// TIA Portal V20 export
FUNCTION "CollectAlarms" : Void   // FC91, LAD
TITLE = Alarm Collector Unit
// Collects alarms from the respective level and categorises the alarms into the different alarm classes.
// stored: Namespace Unit1.Em5, SetENOAutomatically false
   VAR_INPUT
      resetAlarms : Bool;
      disableAlarms : Bool;
   END_VAR
   VAR_OUTPUT
      commandsToUnit : "LUC_typeStateCommands";   // Feedback to the unit
   END_VAR
   VAR CONSTANT
      DelayTime : Time := T#300ms;
      TRUE : Bool := TRUE;
      FALSE : Bool := FALSE;
   END_VAR
BEGIN

REGION Network 1: Reset Alarms
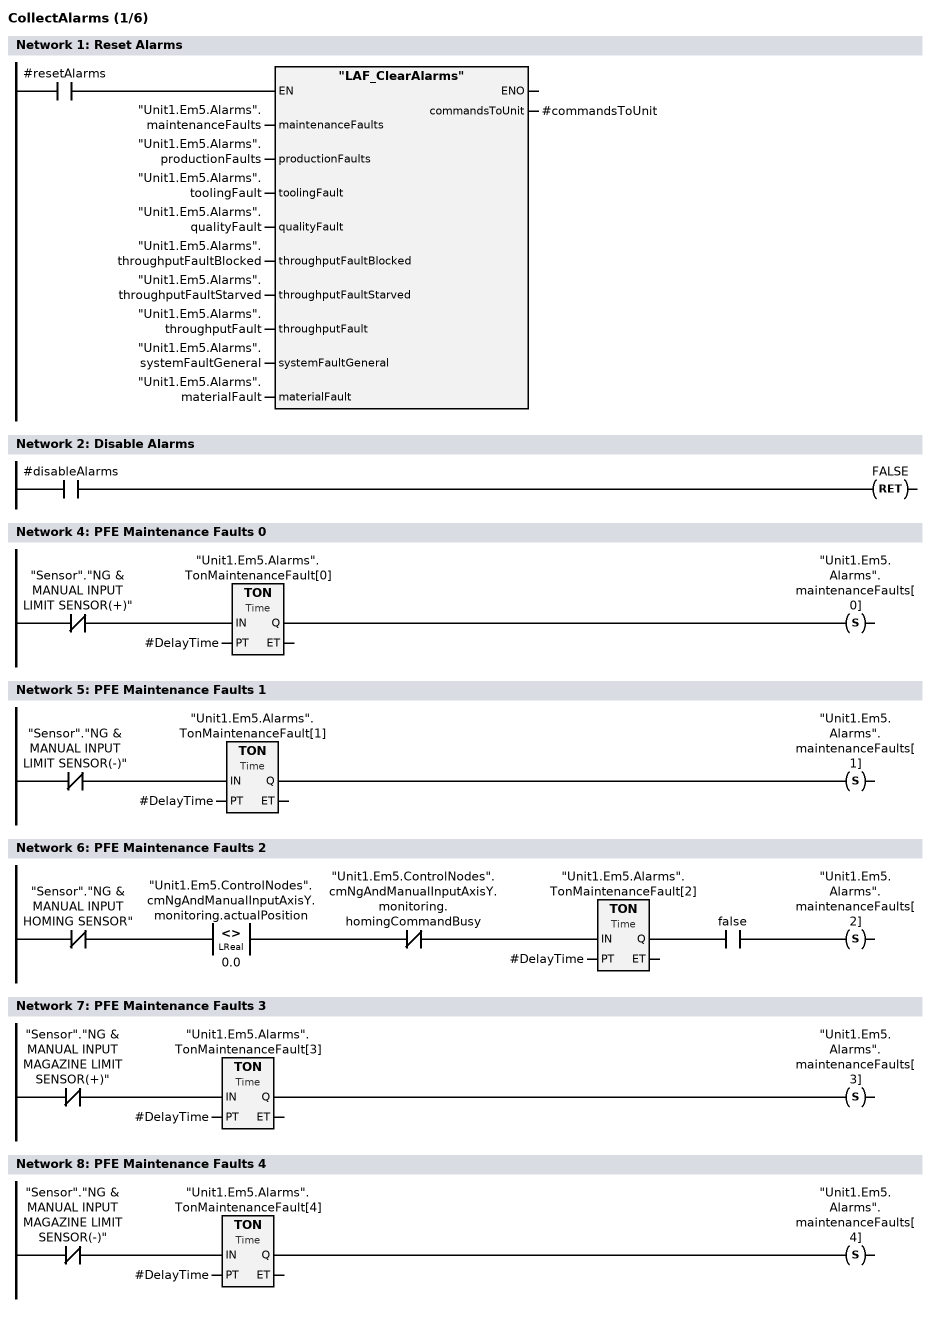
   RUNG wire#powerrail
      Contact( #resetAlarms )
      "LAF_ClearAlarms"(maintenanceFaults := "Unit1.Em5.Alarms".maintenanceFaults, productionFaults := "Unit1.Em5.Alarms".productionFaults, toolingFault := "Unit1.Em5.Alarms".toolingFault, qualityFault := "Unit1.Em5.Alarms".qualityFault, throughputFaultBlocked := "Unit1.Em5.Alarms".throughputFaultBlocked, throughputFaultStarved := "Unit1.Em5.Alarms".throughputFaultStarved, throughputFault := "Unit1.Em5.Alarms".throughputFault, systemFaultGeneral := "Unit1.Em5.Alarms".systemFaultGeneral, materialFault := "Unit1.Em5.Alarms".materialFault, commandsToUnit => #commandsToUnit)
   END_RUNG
   // the same network as SCL:
   IF #resetAlarms THEN
       "LAF_ClearAlarms"(maintenanceFaults := "Unit1.Em5.Alarms".maintenanceFaults,
                         productionFaults := "Unit1.Em5.Alarms".productionFaults,
                         toolingFault := "Unit1.Em5.Alarms".toolingFault,
                         qualityFault := "Unit1.Em5.Alarms".qualityFault,
                         throughputFaultBlocked := "Unit1.Em5.Alarms".throughputFaultBlocked,
                         throughputFaultStarved := "Unit1.Em5.Alarms".throughputFaultStarved,
                         throughputFault := "Unit1.Em5.Alarms".throughputFault,
                         systemFaultGeneral := "Unit1.Em5.Alarms".systemFaultGeneral,
                         materialFault := "Unit1.Em5.Alarms".materialFault,
                         commandsToUnit => #commandsToUnit);
   END_IF;
END_REGION

REGION Network 2: Disable Alarms
   RUNG wire#powerrail
      Contact( #disableAlarms )
      ReturnCoil( FALSE )
   END_RUNG
   // the same network as SCL:
   IF #disableAlarms THEN
       ENO := FALSE;
       RETURN;
   END_IF;
END_REGION

REGION Network 3: *************** Fault ************************
END_REGION

REGION Network 4: PFE Maintenance Faults 0
   RUNG wire#powerrail
      I_Contact( "Sensor"."NG & MANUAL INPUT LIMIT SENSOR(+)" )
      { S7_Templates := "time_type := Time" } "Unit1.Em5.Alarms".TonMaintenanceFault[0].TON(pt := #DelayTime, et =>)
      S_Coil( "Unit1.Em5.Alarms".maintenanceFaults[0] )
   END_RUNG
   // the same network as SCL:
   "Unit1.Em5.Alarms".TonMaintenanceFault[0].TON(IN := NOT "Sensor"."NG & MANUAL INPUT LIMIT SENSOR(+)",
                           PT := #DelayTime);
   IF "Unit1.Em5.Alarms".TonMaintenanceFault[0].Q THEN
       "Unit1.Em5.Alarms".maintenanceFaults[0] := TRUE;
   END_IF;
END_REGION

REGION Network 5: PFE Maintenance Faults 1
   RUNG wire#powerrail
      I_Contact( "Sensor"."NG & MANUAL INPUT LIMIT SENSOR(-)" )
      { S7_Templates := "time_type := Time" } "Unit1.Em5.Alarms".TonMaintenanceFault[1].TON(pt := #DelayTime, et =>)
      S_Coil( "Unit1.Em5.Alarms".maintenanceFaults[1] )
   END_RUNG
   // the same network as SCL:
   "Unit1.Em5.Alarms".TonMaintenanceFault[1].TON(IN := NOT "Sensor"."NG & MANUAL INPUT LIMIT SENSOR(-)",
                           PT := #DelayTime);
   IF "Unit1.Em5.Alarms".TonMaintenanceFault[1].Q THEN
       "Unit1.Em5.Alarms".maintenanceFaults[1] := TRUE;
   END_IF;
END_REGION

REGION Network 6: PFE Maintenance Faults 2
   RUNG wire#powerrail
      I_Contact( "Sensor"."NG & MANUAL INPUT HOMING SENSOR" )
      { S7_Templates := "SrcType := LReal" } NE_Contact(in1 := "Unit1.Em5.ControlNodes".cmNgAndManualInputAxisY.monitoring.actualPosition, in2 := 0.0)
      I_Contact( "Unit1.Em5.ControlNodes".cmNgAndManualInputAxisY.monitoring.homingCommandBusy )
      { S7_Templates := "time_type := Time" } "Unit1.Em5.Alarms".TonMaintenanceFault[2].TON(pt := #DelayTime, et =>)
      Contact( false )
      S_Coil( "Unit1.Em5.Alarms".maintenanceFaults[2] )
   END_RUNG
   // the same network as SCL:
   "Unit1.Em5.Alarms".TonMaintenanceFault[2].TON(IN := NOT "Sensor"."NG & MANUAL INPUT HOMING SENSOR" AND ("Unit1.Em5.ControlNodes".cmNgAndManualInputAxisY.monitoring.actualPosition <> 0.0) AND NOT "Unit1.Em5.ControlNodes".cmNgAndManualInputAxisY.monitoring.homingCommandBusy,
                           PT := #DelayTime);
   IF "Unit1.Em5.Alarms".TonMaintenanceFault[2].Q AND false THEN
       "Unit1.Em5.Alarms".maintenanceFaults[2] := TRUE;
   END_IF;
END_REGION

REGION Network 7: PFE Maintenance Faults 3
   RUNG wire#powerrail
      I_Contact( "Sensor"."NG & MANUAL INPUT MAGAZINE LIMIT SENSOR(+)" )
      { S7_Templates := "time_type := Time" } "Unit1.Em5.Alarms".TonMaintenanceFault[3].TON(pt := #DelayTime, et =>)
      S_Coil( "Unit1.Em5.Alarms".maintenanceFaults[3] )
   END_RUNG
   // the same network as SCL:
   "Unit1.Em5.Alarms".TonMaintenanceFault[3].TON(IN := NOT "Sensor"."NG & MANUAL INPUT MAGAZINE LIMIT SENSOR(+)",
                           PT := #DelayTime);
   IF "Unit1.Em5.Alarms".TonMaintenanceFault[3].Q THEN
       "Unit1.Em5.Alarms".maintenanceFaults[3] := TRUE;
   END_IF;
END_REGION

REGION Network 8: PFE Maintenance Faults 4
   RUNG wire#powerrail
      I_Contact( "Sensor"."NG & MANUAL INPUT MAGAZINE LIMIT SENSOR(-)" )
      { S7_Templates := "time_type := Time" } "Unit1.Em5.Alarms".TonMaintenanceFault[4].TON(pt := #DelayTime, et =>)
      S_Coil( "Unit1.Em5.Alarms".maintenanceFaults[4] )
   END_RUNG
   // the same network as SCL:
   "Unit1.Em5.Alarms".TonMaintenanceFault[4].TON(IN := NOT "Sensor"."NG & MANUAL INPUT MAGAZINE LIMIT SENSOR(-)",
                           PT := #DelayTime);
   IF "Unit1.Em5.Alarms".TonMaintenanceFault[4].Q THEN
       "Unit1.Em5.Alarms".maintenanceFaults[4] := TRUE;
   END_IF;
END_REGION

REGION Network 9: PFE Maintenance Faults 5
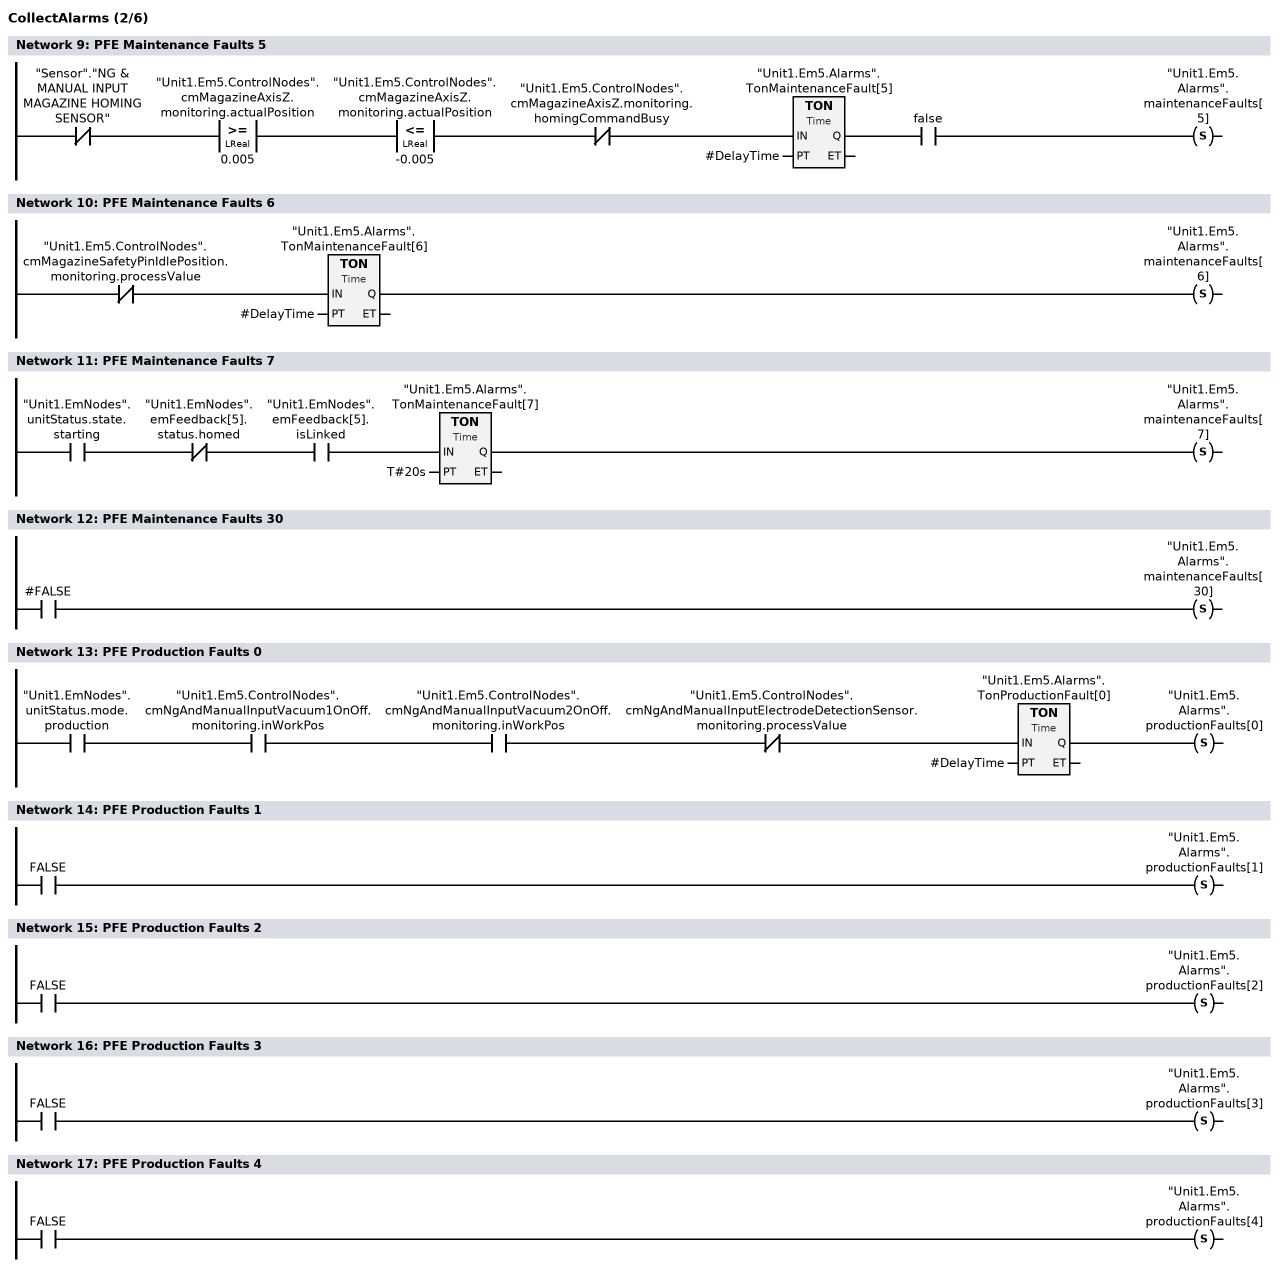
   RUNG wire#powerrail
      I_Contact( "Sensor"."NG & MANUAL INPUT MAGAZINE HOMING SENSOR" )
      { S7_Templates := "SrcType := LReal" } GE_Contact(in1 := "Unit1.Em5.ControlNodes".cmMagazineAxisZ.monitoring.actualPosition, in2 := 0.005)
      { S7_Templates := "SrcType := LReal" } LE_Contact(in1 := "Unit1.Em5.ControlNodes".cmMagazineAxisZ.monitoring.actualPosition, in2 := -0.005)
      I_Contact( "Unit1.Em5.ControlNodes".cmMagazineAxisZ.monitoring.homingCommandBusy )
      { S7_Templates := "time_type := Time" } "Unit1.Em5.Alarms".TonMaintenanceFault[5].TON(pt := #DelayTime, et =>)
      Contact( false )
      S_Coil( "Unit1.Em5.Alarms".maintenanceFaults[5] )
   END_RUNG
   // the same network as SCL:
   "Unit1.Em5.Alarms".TonMaintenanceFault[5].TON(IN := NOT "Sensor"."NG & MANUAL INPUT MAGAZINE HOMING SENSOR" AND ("Unit1.Em5.ControlNodes".cmMagazineAxisZ.monitoring.actualPosition >= 0.005) AND ("Unit1.Em5.ControlNodes".cmMagazineAxisZ.monitoring.actualPosition <= (-0.005)) AND NOT "Unit1.Em5.ControlNodes".cmMagazineAxisZ.monitoring.homingCommandBusy,
                           PT := #DelayTime);
   IF "Unit1.Em5.Alarms".TonMaintenanceFault[5].Q AND false THEN
       "Unit1.Em5.Alarms".maintenanceFaults[5] := TRUE;
   END_IF;
END_REGION

REGION Network 10: PFE Maintenance Faults 6
   RUNG wire#powerrail
      I_Contact( "Unit1.Em5.ControlNodes".cmMagazineSafetyPinIdlePosition.monitoring.processValue )
      { S7_Templates := "time_type := Time" } "Unit1.Em5.Alarms".TonMaintenanceFault[6].TON(pt := #DelayTime, et =>)
      S_Coil( "Unit1.Em5.Alarms".maintenanceFaults[6] )
   END_RUNG
   // the same network as SCL:
   "Unit1.Em5.Alarms".TonMaintenanceFault[6].TON(IN := NOT "Unit1.Em5.ControlNodes".cmMagazineSafetyPinIdlePosition.monitoring.processValue,
                           PT := #DelayTime);
   IF "Unit1.Em5.Alarms".TonMaintenanceFault[6].Q THEN
       "Unit1.Em5.Alarms".maintenanceFaults[6] := TRUE;
   END_IF;
END_REGION

REGION Network 11: PFE Maintenance Faults 7
   RUNG wire#powerrail
      Contact( "Unit1.EmNodes".unitStatus.state.starting )
      I_Contact( "Unit1.EmNodes".emFeedback[5].status.homed )
      Contact( "Unit1.EmNodes".emFeedback[5].isLinked )
      { S7_Templates := "time_type := Time" } "Unit1.Em5.Alarms".TonMaintenanceFault[7].TON(pt := T#20s, et =>)
      S_Coil( "Unit1.Em5.Alarms".maintenanceFaults[7] )
   END_RUNG
   // the same network as SCL:
   "Unit1.Em5.Alarms".TonMaintenanceFault[7].TON(IN := "Unit1.EmNodes".unitStatus.state.starting AND NOT "Unit1.EmNodes".emFeedback[5].status.homed AND "Unit1.EmNodes".emFeedback[5].isLinked,
                           PT := T#20s);
   IF "Unit1.Em5.Alarms".TonMaintenanceFault[7].Q THEN
       "Unit1.Em5.Alarms".maintenanceFaults[7] := TRUE;
   END_IF;
END_REGION

REGION Network 12: PFE Maintenance Faults 30
   RUNG wire#powerrail
      Contact( #FALSE )
      S_Coil( "Unit1.Em5.Alarms".maintenanceFaults[30] )
   END_RUNG
   // the same network as SCL:
   IF #FALSE THEN "Unit1.Em5.Alarms".maintenanceFaults[30] := TRUE; END_IF;
END_REGION

REGION Network 13: PFE Production Faults 0
   RUNG wire#powerrail
      Contact( "Unit1.EmNodes".unitStatus.mode.production )
      Contact( "Unit1.Em5.ControlNodes".cmNgAndManualInputVacuum1OnOff.monitoring.inWorkPos )
      Contact( "Unit1.Em5.ControlNodes".cmNgAndManualInputVacuum2OnOff.monitoring.inWorkPos )
      I_Contact( "Unit1.Em5.ControlNodes".cmNgAndManualInputElectrodeDetectionSensor.monitoring.processValue )
      { S7_Templates := "time_type := Time" } "Unit1.Em5.Alarms".TonProductionFault[0].TON(pt := #DelayTime, et =>)
      S_Coil( "Unit1.Em5.Alarms".productionFaults[0] )
   END_RUNG
   // the same network as SCL:
   "Unit1.Em5.Alarms".TonProductionFault[0].TON(IN := "Unit1.EmNodes".unitStatus.mode.production AND "Unit1.Em5.ControlNodes".cmNgAndManualInputVacuum1OnOff.monitoring.inWorkPos AND "Unit1.Em5.ControlNodes".cmNgAndManualInputVacuum2OnOff.monitoring.inWorkPos AND NOT "Unit1.Em5.ControlNodes".cmNgAndManualInputElectrodeDetectionSensor.monitoring.processValue,
                           PT := #DelayTime);
   IF "Unit1.Em5.Alarms".TonProductionFault[0].Q THEN "Unit1.Em5.Alarms".productionFaults[0] := TRUE; END_IF;
END_REGION

REGION Network 14: PFE Production Faults 1
   RUNG wire#powerrail
      Contact( FALSE )
      S_Coil( "Unit1.Em5.Alarms".productionFaults[1] )
   END_RUNG
   // the same network as SCL:
   IF FALSE THEN "Unit1.Em5.Alarms".productionFaults[1] := TRUE; END_IF;
END_REGION

REGION Network 15: PFE Production Faults 2
   RUNG wire#powerrail
      Contact( FALSE )
      S_Coil( "Unit1.Em5.Alarms".productionFaults[2] )
   END_RUNG
   // the same network as SCL:
   IF FALSE THEN "Unit1.Em5.Alarms".productionFaults[2] := TRUE; END_IF;
END_REGION

REGION Network 16: PFE Production Faults 3
   RUNG wire#powerrail
      Contact( FALSE )
      S_Coil( "Unit1.Em5.Alarms".productionFaults[3] )
   END_RUNG
   // the same network as SCL:
   IF FALSE THEN "Unit1.Em5.Alarms".productionFaults[3] := TRUE; END_IF;
END_REGION

REGION Network 17: PFE Production Faults 4
   RUNG wire#powerrail
      Contact( FALSE )
      S_Coil( "Unit1.Em5.Alarms".productionFaults[4] )
   END_RUNG
   // the same network as SCL:
   IF FALSE THEN "Unit1.Em5.Alarms".productionFaults[4] := TRUE; END_IF;
END_REGION

REGION Network 18: PFE Tooling Faults 0
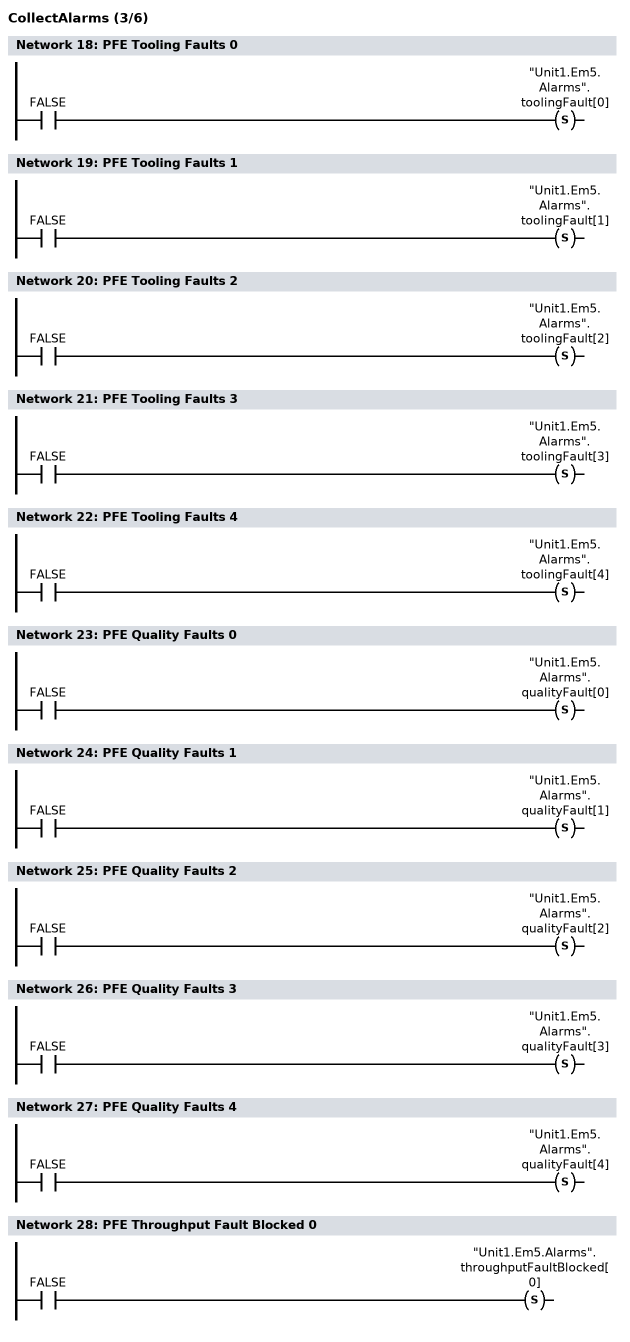
   RUNG wire#powerrail
      Contact( FALSE )
      S_Coil( "Unit1.Em5.Alarms".toolingFault[0] )
   END_RUNG
   // the same network as SCL:
   IF FALSE THEN "Unit1.Em5.Alarms".toolingFault[0] := TRUE; END_IF;
END_REGION

REGION Network 19: PFE Tooling Faults 1
   RUNG wire#powerrail
      Contact( FALSE )
      S_Coil( "Unit1.Em5.Alarms".toolingFault[1] )
   END_RUNG
   // the same network as SCL:
   IF FALSE THEN "Unit1.Em5.Alarms".toolingFault[1] := TRUE; END_IF;
END_REGION

REGION Network 20: PFE Tooling Faults 2
   RUNG wire#powerrail
      Contact( FALSE )
      S_Coil( "Unit1.Em5.Alarms".toolingFault[2] )
   END_RUNG
   // the same network as SCL:
   IF FALSE THEN "Unit1.Em5.Alarms".toolingFault[2] := TRUE; END_IF;
END_REGION

REGION Network 21: PFE Tooling Faults 3
   RUNG wire#powerrail
      Contact( FALSE )
      S_Coil( "Unit1.Em5.Alarms".toolingFault[3] )
   END_RUNG
   // the same network as SCL:
   IF FALSE THEN "Unit1.Em5.Alarms".toolingFault[3] := TRUE; END_IF;
END_REGION

REGION Network 22: PFE Tooling Faults 4
   RUNG wire#powerrail
      Contact( FALSE )
      S_Coil( "Unit1.Em5.Alarms".toolingFault[4] )
   END_RUNG
   // the same network as SCL:
   IF FALSE THEN "Unit1.Em5.Alarms".toolingFault[4] := TRUE; END_IF;
END_REGION

REGION Network 23: PFE Quality Faults 0
   RUNG wire#powerrail
      Contact( FALSE )
      S_Coil( "Unit1.Em5.Alarms".qualityFault[0] )
   END_RUNG
   // the same network as SCL:
   IF FALSE THEN "Unit1.Em5.Alarms".qualityFault[0] := TRUE; END_IF;
END_REGION

REGION Network 24: PFE Quality Faults 1
   RUNG wire#powerrail
      Contact( FALSE )
      S_Coil( "Unit1.Em5.Alarms".qualityFault[1] )
   END_RUNG
   // the same network as SCL:
   IF FALSE THEN "Unit1.Em5.Alarms".qualityFault[1] := TRUE; END_IF;
END_REGION

REGION Network 25: PFE Quality Faults 2
   RUNG wire#powerrail
      Contact( FALSE )
      S_Coil( "Unit1.Em5.Alarms".qualityFault[2] )
   END_RUNG
   // the same network as SCL:
   IF FALSE THEN "Unit1.Em5.Alarms".qualityFault[2] := TRUE; END_IF;
END_REGION

REGION Network 26: PFE Quality Faults 3
   RUNG wire#powerrail
      Contact( FALSE )
      S_Coil( "Unit1.Em5.Alarms".qualityFault[3] )
   END_RUNG
   // the same network as SCL:
   IF FALSE THEN "Unit1.Em5.Alarms".qualityFault[3] := TRUE; END_IF;
END_REGION

REGION Network 27: PFE Quality Faults 4
   RUNG wire#powerrail
      Contact( FALSE )
      S_Coil( "Unit1.Em5.Alarms".qualityFault[4] )
   END_RUNG
   // the same network as SCL:
   IF FALSE THEN "Unit1.Em5.Alarms".qualityFault[4] := TRUE; END_IF;
END_REGION

REGION Network 28: PFE Throughput Fault Blocked 0
   RUNG wire#powerrail
      Contact( FALSE )
      S_Coil( "Unit1.Em5.Alarms".throughputFaultBlocked[0] )
   END_RUNG
   // the same network as SCL:
   IF FALSE THEN "Unit1.Em5.Alarms".throughputFaultBlocked[0] := TRUE; END_IF;
END_REGION

REGION Network 29: PFE Throughput Fault Blocked 1
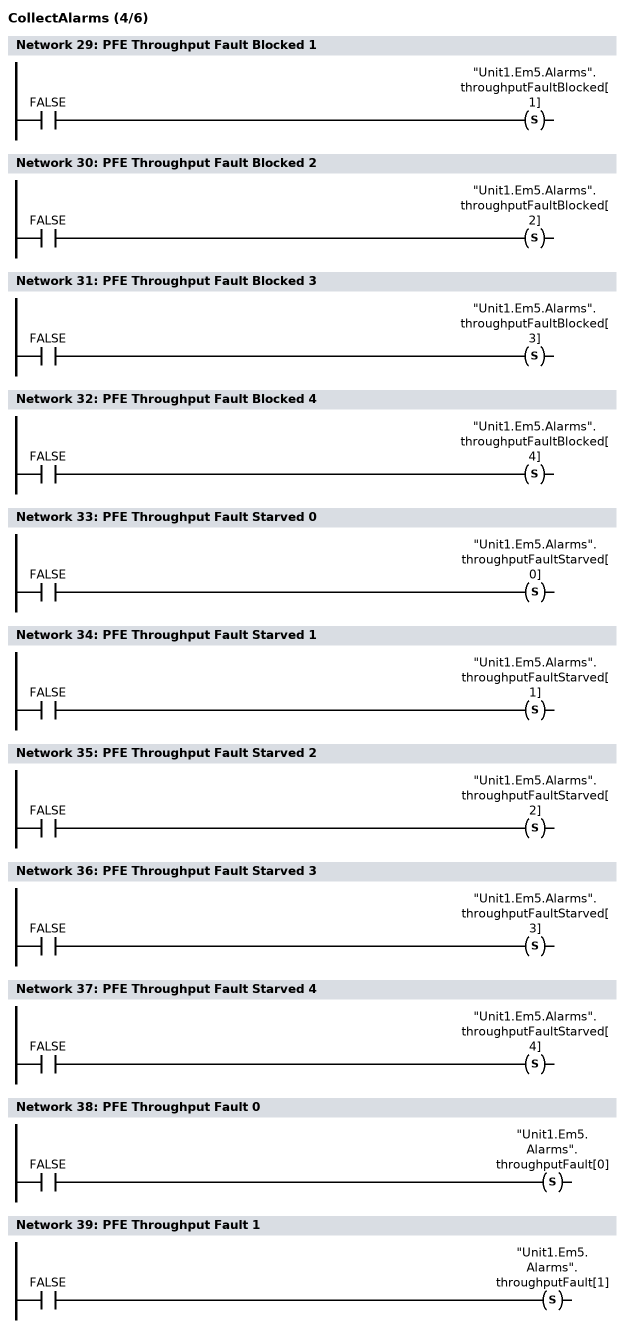
   RUNG wire#powerrail
      Contact( FALSE )
      S_Coil( "Unit1.Em5.Alarms".throughputFaultBlocked[1] )
   END_RUNG
   // the same network as SCL:
   IF FALSE THEN "Unit1.Em5.Alarms".throughputFaultBlocked[1] := TRUE; END_IF;
END_REGION

REGION Network 30: PFE Throughput Fault Blocked 2
   RUNG wire#powerrail
      Contact( FALSE )
      S_Coil( "Unit1.Em5.Alarms".throughputFaultBlocked[2] )
   END_RUNG
   // the same network as SCL:
   IF FALSE THEN "Unit1.Em5.Alarms".throughputFaultBlocked[2] := TRUE; END_IF;
END_REGION

REGION Network 31: PFE Throughput Fault Blocked 3
   RUNG wire#powerrail
      Contact( FALSE )
      S_Coil( "Unit1.Em5.Alarms".throughputFaultBlocked[3] )
   END_RUNG
   // the same network as SCL:
   IF FALSE THEN "Unit1.Em5.Alarms".throughputFaultBlocked[3] := TRUE; END_IF;
END_REGION

REGION Network 32: PFE Throughput Fault Blocked 4
   RUNG wire#powerrail
      Contact( FALSE )
      S_Coil( "Unit1.Em5.Alarms".throughputFaultBlocked[4] )
   END_RUNG
   // the same network as SCL:
   IF FALSE THEN "Unit1.Em5.Alarms".throughputFaultBlocked[4] := TRUE; END_IF;
END_REGION

REGION Network 33: PFE Throughput Fault Starved 0
   RUNG wire#powerrail
      Contact( FALSE )
      S_Coil( "Unit1.Em5.Alarms".throughputFaultStarved[0] )
   END_RUNG
   // the same network as SCL:
   IF FALSE THEN "Unit1.Em5.Alarms".throughputFaultStarved[0] := TRUE; END_IF;
END_REGION

REGION Network 34: PFE Throughput Fault Starved 1
   RUNG wire#powerrail
      Contact( FALSE )
      S_Coil( "Unit1.Em5.Alarms".throughputFaultStarved[1] )
   END_RUNG
   // the same network as SCL:
   IF FALSE THEN "Unit1.Em5.Alarms".throughputFaultStarved[1] := TRUE; END_IF;
END_REGION

REGION Network 35: PFE Throughput Fault Starved 2
   RUNG wire#powerrail
      Contact( FALSE )
      S_Coil( "Unit1.Em5.Alarms".throughputFaultStarved[2] )
   END_RUNG
   // the same network as SCL:
   IF FALSE THEN "Unit1.Em5.Alarms".throughputFaultStarved[2] := TRUE; END_IF;
END_REGION

REGION Network 36: PFE Throughput Fault Starved 3
   RUNG wire#powerrail
      Contact( FALSE )
      S_Coil( "Unit1.Em5.Alarms".throughputFaultStarved[3] )
   END_RUNG
   // the same network as SCL:
   IF FALSE THEN "Unit1.Em5.Alarms".throughputFaultStarved[3] := TRUE; END_IF;
END_REGION

REGION Network 37: PFE Throughput Fault Starved 4
   RUNG wire#powerrail
      Contact( FALSE )
      S_Coil( "Unit1.Em5.Alarms".throughputFaultStarved[4] )
   END_RUNG
   // the same network as SCL:
   IF FALSE THEN "Unit1.Em5.Alarms".throughputFaultStarved[4] := TRUE; END_IF;
END_REGION

REGION Network 38: PFE Throughput Fault 0
   RUNG wire#powerrail
      Contact( FALSE )
      S_Coil( "Unit1.Em5.Alarms".throughputFault[0] )
   END_RUNG
   // the same network as SCL:
   IF FALSE THEN "Unit1.Em5.Alarms".throughputFault[0] := TRUE; END_IF;
END_REGION

REGION Network 39: PFE Throughput Fault 1
   RUNG wire#powerrail
      Contact( FALSE )
      S_Coil( "Unit1.Em5.Alarms".throughputFault[1] )
   END_RUNG
   // the same network as SCL:
   IF FALSE THEN "Unit1.Em5.Alarms".throughputFault[1] := TRUE; END_IF;
END_REGION

REGION Network 40: PFE Throughput Fault 2
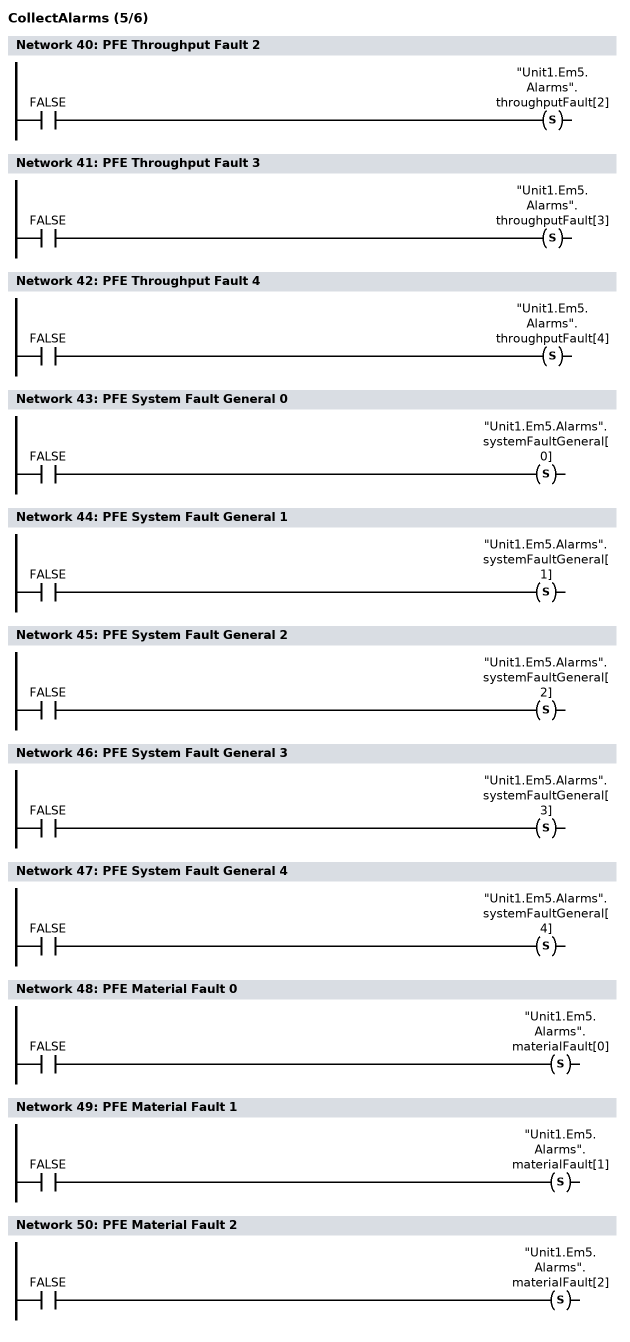
   RUNG wire#powerrail
      Contact( FALSE )
      S_Coil( "Unit1.Em5.Alarms".throughputFault[2] )
   END_RUNG
   // the same network as SCL:
   IF FALSE THEN "Unit1.Em5.Alarms".throughputFault[2] := TRUE; END_IF;
END_REGION

REGION Network 41: PFE Throughput Fault 3
   RUNG wire#powerrail
      Contact( FALSE )
      S_Coil( "Unit1.Em5.Alarms".throughputFault[3] )
   END_RUNG
   // the same network as SCL:
   IF FALSE THEN "Unit1.Em5.Alarms".throughputFault[3] := TRUE; END_IF;
END_REGION

REGION Network 42: PFE Throughput Fault 4
   RUNG wire#powerrail
      Contact( FALSE )
      S_Coil( "Unit1.Em5.Alarms".throughputFault[4] )
   END_RUNG
   // the same network as SCL:
   IF FALSE THEN "Unit1.Em5.Alarms".throughputFault[4] := TRUE; END_IF;
END_REGION

REGION Network 43: PFE System Fault General 0
   RUNG wire#powerrail
      Contact( FALSE )
      S_Coil( "Unit1.Em5.Alarms".systemFaultGeneral[0] )
   END_RUNG
   // the same network as SCL:
   IF FALSE THEN "Unit1.Em5.Alarms".systemFaultGeneral[0] := TRUE; END_IF;
END_REGION

REGION Network 44: PFE System Fault General 1
   RUNG wire#powerrail
      Contact( FALSE )
      S_Coil( "Unit1.Em5.Alarms".systemFaultGeneral[1] )
   END_RUNG
   // the same network as SCL:
   IF FALSE THEN "Unit1.Em5.Alarms".systemFaultGeneral[1] := TRUE; END_IF;
END_REGION

REGION Network 45: PFE System Fault General 2
   RUNG wire#powerrail
      Contact( FALSE )
      S_Coil( "Unit1.Em5.Alarms".systemFaultGeneral[2] )
   END_RUNG
   // the same network as SCL:
   IF FALSE THEN "Unit1.Em5.Alarms".systemFaultGeneral[2] := TRUE; END_IF;
END_REGION

REGION Network 46: PFE System Fault General 3
   RUNG wire#powerrail
      Contact( FALSE )
      S_Coil( "Unit1.Em5.Alarms".systemFaultGeneral[3] )
   END_RUNG
   // the same network as SCL:
   IF FALSE THEN "Unit1.Em5.Alarms".systemFaultGeneral[3] := TRUE; END_IF;
END_REGION

REGION Network 47: PFE System Fault General 4
   RUNG wire#powerrail
      Contact( FALSE )
      S_Coil( "Unit1.Em5.Alarms".systemFaultGeneral[4] )
   END_RUNG
   // the same network as SCL:
   IF FALSE THEN "Unit1.Em5.Alarms".systemFaultGeneral[4] := TRUE; END_IF;
END_REGION

REGION Network 48: PFE Material Fault 0
   RUNG wire#powerrail
      Contact( FALSE )
      S_Coil( "Unit1.Em5.Alarms".materialFault[0] )
   END_RUNG
   // the same network as SCL:
   IF FALSE THEN "Unit1.Em5.Alarms".materialFault[0] := TRUE; END_IF;
END_REGION

REGION Network 49: PFE Material Fault 1
   RUNG wire#powerrail
      Contact( FALSE )
      S_Coil( "Unit1.Em5.Alarms".materialFault[1] )
   END_RUNG
   // the same network as SCL:
   IF FALSE THEN "Unit1.Em5.Alarms".materialFault[1] := TRUE; END_IF;
END_REGION

REGION Network 50: PFE Material Fault 2
   RUNG wire#powerrail
      Contact( FALSE )
      S_Coil( "Unit1.Em5.Alarms".materialFault[2] )
   END_RUNG
   // the same network as SCL:
   IF FALSE THEN "Unit1.Em5.Alarms".materialFault[2] := TRUE; END_IF;
END_REGION

REGION Network 51: PFE Material Fault 3
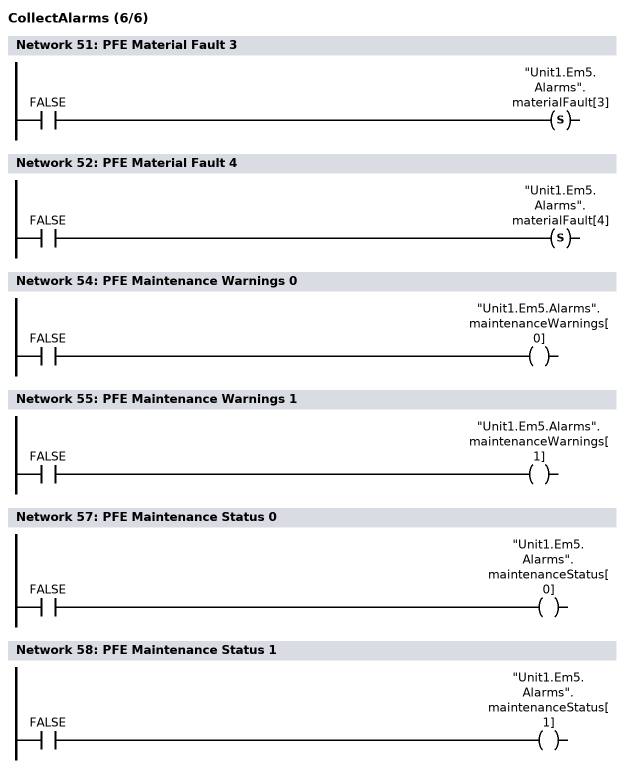
   RUNG wire#powerrail
      Contact( FALSE )
      S_Coil( "Unit1.Em5.Alarms".materialFault[3] )
   END_RUNG
   // the same network as SCL:
   IF FALSE THEN "Unit1.Em5.Alarms".materialFault[3] := TRUE; END_IF;
END_REGION

REGION Network 52: PFE Material Fault 4
   RUNG wire#powerrail
      Contact( FALSE )
      S_Coil( "Unit1.Em5.Alarms".materialFault[4] )
   END_RUNG
   // the same network as SCL:
   IF FALSE THEN "Unit1.Em5.Alarms".materialFault[4] := TRUE; END_IF;
END_REGION

REGION Network 53: *************** Warning **************************
END_REGION

REGION Network 54: PFE Maintenance Warnings 0
   RUNG wire#powerrail
      Contact( FALSE )
      Coil( "Unit1.Em5.Alarms".maintenanceWarnings[0] )
   END_RUNG
   // the same network as SCL:
   "Unit1.Em5.Alarms".maintenanceWarnings[0] := FALSE;
END_REGION

REGION Network 55: PFE Maintenance Warnings 1
   RUNG wire#powerrail
      Contact( FALSE )
      Coil( "Unit1.Em5.Alarms".maintenanceWarnings[1] )
   END_RUNG
   // the same network as SCL:
   "Unit1.Em5.Alarms".maintenanceWarnings[1] := FALSE;
END_REGION

REGION Network 56: *************** Status ***************************
END_REGION

REGION Network 57: PFE Maintenance Status 0
   RUNG wire#powerrail
      Contact( FALSE )
      Coil( "Unit1.Em5.Alarms".maintenanceStatus[0] )
   END_RUNG
   // the same network as SCL:
   "Unit1.Em5.Alarms".maintenanceStatus[0] := FALSE;
END_REGION

REGION Network 58: PFE Maintenance Status 1
   RUNG wire#powerrail
      Contact( FALSE )
      Coil( "Unit1.Em5.Alarms".maintenanceStatus[1] )
   END_RUNG
   // the same network as SCL:
   "Unit1.Em5.Alarms".maintenanceStatus[1] := FALSE;
END_REGION
END_FUNCTION
